// LS Electric XG5000 project: DAY16
// PLC LSPLC
// module base 0 slot 0: 입출력 모듈:XBC-DR30S (DC 24V 입력 18점, 릴레이 출력 12점)

PROGRAM DAY16 (task: 스캔 프로그램)

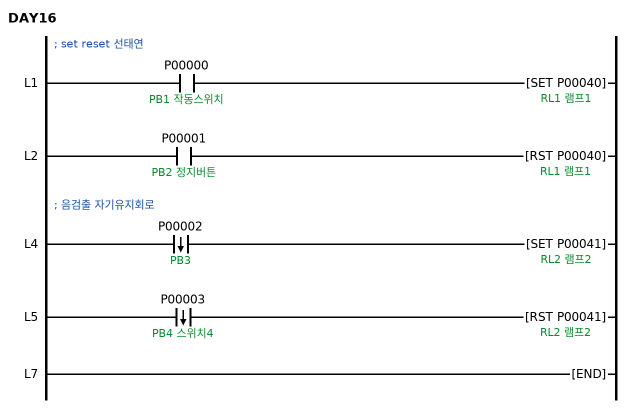
// set reset 선태연
; L1
LOAD      P00000	// PB1 작동스위치
SET       P00040	// RL1 램프1
; L2
LOAD      P00001	// PB2 정지버튼
RST       P00040	// RL1 램프1
// 음검출 자기유지회로
; L4
LOADN     P00002	// PB3
SET       P00041	// RL2 램프2
; L5
LOADN     P00003	// PB4 스위치4
RST       P00041	// RL2 램프2
; L7
END